// TIA Portal V20 export
TYPE "LER_typeAlignCalibrationInterface"
// stored: Access Published
   STRUCT
      commands : "LER_typeAlignCalibrationCommands";
      monitoring : "LER_typeAlignCalibrationMonitoring";
      configuration : "LER_typeAlignCalibrationConfiguration";
   END_STRUCT;
END_TYPE
